FUNCTION_BLOCK DM_KRMT (* Remote Device Management Kernel *)
  (* Standard: 61499 Demo ITA; Function: Device Management; Description: Remote Device Management Kernel *)
  (* Version 0.2, 2008-06-04, JHC, Holobloc Inc, Updated DOCTYPE. *)
  (* Version 0.1, 2001-01-21, JHC, Rockwell Automation, Modified per new DM_CLT service spec *)
  (* Version 0.0, 2000-12-31, JHC, Rockwell Automation, Initial version *)
  (* Compiler header: package fb.rt; import fb.rt.net.*; *)
  (* Compiler Java IBM VisualAge 3.0 *)
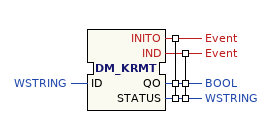
  EVENT_OUTPUT
    INITO WITH QO, STATUS; (* Initialize/Terminate Confirmation *)
    IND WITH QO, STATUS; (* Message Arrival *)
  END_EVENT
  VAR_INPUT
    ID : WSTRING := "localhost:61499"; (* Server ID *)
  END_VAR
  VAR_OUTPUT
    QO : BOOL; (* 1=Initiated,0=Terminated *)
    STATUS : WSTRING; (* "OK"or Reason for Termination *)
  END_VAR
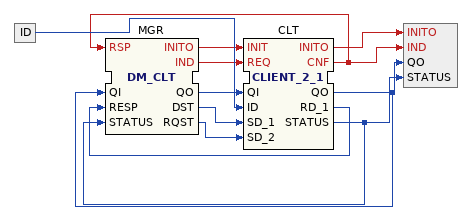
  FBS
    CLT : CLIENT_2_1;
    MGR : DM_CLT;
  END_FBS
  EVENT_CONNECTIONS
    MGR.INITO TO CLT.INIT;
    MGR.IND TO CLT.REQ;
    CLT.INITO TO INITO;
    CLT.CNF TO MGR.RSP;
    CLT.CNF TO IND;
  END_CONNECTIONS
  DATA_CONNECTIONS
    MGR.QO TO CLT.QI;
    CLT.QO TO MGR.QI;
    CLT.QO TO QO;
    ID TO CLT.ID;
    MGR.DST TO CLT.SD_1;
    MGR.RQST TO CLT.SD_2;
    CLT.RD_1 TO MGR.RESP;
    CLT.STATUS TO MGR.STATUS;
    CLT.STATUS TO STATUS;
  END_CONNECTIONS
END_FUNCTION_BLOCK
